// TwinCAT 3 PLC project PLC
// ProgramVersion: 3.1.4026.19
// CompilerDefines: VISU_USEPROPERTYINFO
// libraries:
//   Tc2_Standard, * (Beckhoff Automation GmbH)
//   Tc2_System, * (Beckhoff Automation GmbH)
// project tree:
//   / GlobalTextList.TcGTLO, PlcTask.TcTTO, Visualization Manager.TcVMO (not stored)
//   POUs/ MAIN.TcPOU
//   VISUs/ Visualization.TcVIS
// real-time tasks:
//   TASK PlcTask: cycle T#10ms, priority 20, ADS port 350

CONFIGURATION PLC
    RESOURCE PLC ON TwinCAT3
        TASK PlcTask(INTERVAL := T#10ms, PRIORITY := 20);
        PROGRAM MAIN WITH PlcTask : MAIN;
    END_RESOURCE
END_CONFIGURATION

// ---- POUs/MAIN.TcPOU
PROGRAM MAIN
VAR
	iState : INT := 0;
	bStartButton : BOOL;
	bSensorTop : BOOL := TRUE;
	bSensorBottom : BOOL;
	bPistonDown : BOOL;
	bPistonUp : BOOL;
END_VAR

CASE iState OF
	0:
		bPistonDown := FALSE;
		bPistonUp := FALSE;
		
		IF bStartButton AND bSensorTop THEN
			iState := 10;
		END_IF
		
	10:
		bPistonDown := TRUE;
		bSensorTop := FALSE;
		
		IF bSensorBottom THEN
			bPistonDown := FALSE;
			iState := 20;
		END_IF
		
	20:
		bPistonUp := TRUE;
		bSensorBottom := FALSE;
		
		IF bSensorTop THEN
			bPistonUp := FALSE;
			iState := 0;
		END_IF		
END_CASE

END_PROGRAM

// ---- GlobalTextList.TcGTLO
TEXTLIST GlobalTextList
  996 = 'Piston Down'
  65 = 'Piston Up'
  644 = 'Sensor Bottom'
  89 = 'Sensor Up'
  232 = 'State: %d'
END_TEXTLIST

// ---- VISUs/Visualization.TcVIS
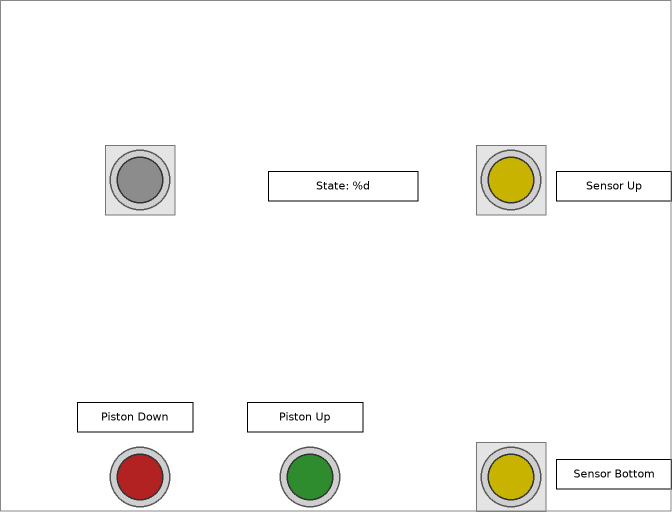
VISUALIZATION Visualization  // 672x512
    PushSwitch (105,145 70x70), variable: MAIN.bStartButton, behaviour: TOGGLE, style: Switch-PushSwitch-Gray
    Lamp1 (105,442 70x70), variable: MAIN.bPistonDown, style: Lamp-Lamp1-Red
    Lamp1 (275,442 70x70), variable: MAIN.bPistonUp, style: Lamp-Lamp1-Green
    Rectangle (268,171 150x30), "State: %d", text variable: MAIN.iState
    Rectangle (77,402 116x30), "Piston Down", text variable: MAIN.iState
    Rectangle (247,402 116x30), "Piston Up", text variable: MAIN.iState
    Rectangle (556,459 116x30), "Sensor Bottom", text variable: MAIN.iState
    Rectangle (556,171 116x30), "Sensor Up", text variable: MAIN.iState
    PushSwitch (476,442 70x70), variable: MAIN.bSensorBottom, behaviour: TOGGLE, style: Switch-PushSwitch-Yellow
    PushSwitch (476,145 70x70), variable: MAIN.bSensorTop, behaviour: TOGGLE, style: Switch-PushSwitch-Yellow
END_VISUALIZATION
